// TIA Portal V19 export
TYPE "LEXCHANGETRAY_typePlasticWorkStationIoSignalInterface"
// configuration: LEXCHANGETRAY_typePlasticWorkStationIoSignalConfigeration
// commands: LEXCHANGETRAY_typePlasticWorkStationIoSignalManualCommands
// monitoring: LEXCHANGETRAY_typePlasticWorkStationIoSignalProcessValues
// stored: Access Published
   STRUCT
      configuration : "LEXCHANGETRAY_typePlasticWorkStationIoSignalConfigeration";
      commands { S7_SetPoint := 'True'} : "LEXCHANGETRAY_typePlasticWorkStationIoSignalManualCommands";
      monitoring { S7_SetPoint := 'True'} : "LEXCHANGETRAY_typePlasticWorkStationIoSignalProcessValues";
   END_STRUCT;
END_TYPE
